{attribute 'GeneratedUsingTerminal: EL9576-0000-0016'}
{attribute addProperty BoxType "EL9576-0000-0016"}
{attribute addProperty Id "BCT_InputsAT %I*BCT_Inputs_28C1780C15WcStateAT %I*WcState_9091E0EB2InfoDataAT %I*InfoData_94A18F5E2"}
{attribute addProperty CRC "3384031510"}
{attribute addProperty Size "19"}
TYPE EL9576_C9B43916 EXTENDS EtcSlaveTerminalBase_947E5A46 :
STRUCT
	{attribute addProperty Name "BCT_Inputs"}
	BCT_Inputs : BCT_Inputs_28C1780C;
	{attribute addProperty Name "WcState"}
	WcState : WcState_9091E0EB;
	{attribute addProperty Name "InfoData"}
	InfoData : InfoData_94A18F5E;
END_STRUCT
END_TYPE

(* stored: Version 1.2.0.0, ProductVersion 3.1.4024.9
   DUT EL9576_C9B43916: Id {08b3acc1-d254-428b-a793-530c15f95f86} *)
